FUNCTION_BLOCK FB_TwinSAFEArm
VAR_INPUT
	bFeedBackEstopOut     	:BOOL;
	bFeedBackSDCIn			:BOOL;
	
END_VAR
VAR_OUTPUT
	bRestartToggle			:BOOL;
	bSDCPrimed 				:BOOL;
END_VAR
VAR
END_VAR

IF NOT bFeedBackEstopOut AND bFeedBackSDCIn THEN
	bRestartToggle := NOT bRestartToggle;
ELSIF bFeedBackEstopOut THEN
	bSDCPrimed := TRUE;
END_IF

END_FUNCTION_BLOCK

(* stored: Version 1.1.0.1
   POU FB_TwinSAFEArm: Id {fea34919-40af-4ef0-81ea-c4ec8124354e}, SpecialFunc None *)
